// TIA Portal V17 export
// export: Created 2021-12-03T08:12:52.8743483Z, ExportSetting WithDefaults, DisplayName Totally Integrated Automation Portal, DisplayVersion V17, DisplayName TIA Portal Openness, DisplayVersion V17, DisplayName TIA Portal Version Control Interface, DisplayVersion V17, DisplayName STEP 7 Professional, DisplayVersion V17, DisplayName STEP 7 Safety, DisplayVersion V17, DisplayName WinCC Advanced, DisplayVersion V17
DATA_BLOCK "GDB_HmiToPlc"   // DB1002
VERSION : 0.1
// stored: AutoNumber false, IsOnlyStoredInLoadMemory false, IsWriteProtectedInAS false
   VAR
      CmndON : Word;   // Команды включения
      CmndOFF : Word;   // Команды отключения
      Cmnd_AckRst : Word;   // Команды сброса
      CmndSwitch : Word;   // Команды переключения
      Service_Button1 : Word;   // Кнопки в сервисном меню
      Service_Button2 : Word;   // Кнопки в сервисном меню
   END_VAR
BEGIN
END_DATA_BLOCK
